FUNCTION_BLOCK POU_1
VAR_INPUT
END_VAR
VAR_OUTPUT
END_VAR
VAR
END_VAR

// NETWORK 1

END_FUNCTION_BLOCK

(* stored: Version 1.1.0.1, ProductVersion 3.1.4024.11
   POU POU_1: Id {c647c264-4cec-4957-bb73-bb44ea2a672a}, SpecialFunc None *)
